{attribute addProperty BoxType "KL2642-0050"}
{attribute addProperty Id "Channel_1Channel_3CF6834E00Channel_2Channel_3CF6834E00"}
{attribute addProperty CRC "422038865"}
{attribute addProperty SizeInBites "0"}
{attribute addProperty SizeInBytes "0"}
TYPE KL_1927CD51 :
STRUCT
	{attribute addProperty Name "Channel_1"}
	Channel_1 : Channel_3CF6834E;
	{attribute addProperty Name "Channel_2"}
	Channel_2 : Channel_3CF6834E;
END_STRUCT
END_TYPE

(* stored: Version 1.2.0.0, ProductVersion 3.1.4024.9
   DUT KL_1927CD51: Id {476128c8-55d3-4dd4-9e90-a00603734b9e} *)
